FUNCTION_BLOCK LoadGraphRpcHandler IMPLEMENTS I_RpcHandler
VAR
	graph : I_Graph;
END_VAR

METHOD FB_init : BOOL
VAR_INPUT
	bInitRetains : BOOL; // if TRUE, the retain variables are initialized (warm start / cold start)
	bInCopyCode : BOOL;  // if TRUE, the instance afterwards gets moved into the copy code (online change)
	Graph : I_Graph;
END_VAR
this^.graph := Graph;
END_METHOD

METHOD Handle
VAR_INPUT
	Parameters : I_Deserializer;
	Response : I_SynchronousRpcResponse;
END_VAR
VAR
	feedback : DeserializerFeedback;
	graphDeserializer : I_Deserializer;
END_VAR
graphDeserializer := Parameters.GetKeyObject('graph');

IF NOT graph.TryDeserializeFrom(graphDeserializer, feedback) THEN
	Response.RejectWithMessage(feedback.FirstError.Message);
END_IF

Response.CompleteWithObject(graph);
END_METHOD

END_FUNCTION_BLOCK

(* stored: Version 1.1.0.1, ProductVersion 3.1.4024.12
   POU LoadGraphRpcHandler: Id {d7516374-45eb-4b62-8de2-ab2fefa44ac4}, SpecialFunc None
   Folder Constructor: Id {ff32cb99-3e6f-4c6a-aa11-5015f7dccc68}
   Method FB_init: Id {11b3e155-9572-4842-9264-53fd7e33eefe}
   Method Handle: Id {eccafacb-820d-475e-bb11-2e1cd4050d86} *)
